FUNCTION_BLOCK MUX_DWORD (* See MUX_ANY *)
  (* Standard: 61131-3 *)
  (* Version 0.0, 2004-12-15, JHC, Rockwell Automation, Converted from SRC format. *)
  (* Compiler header: package fb.rt.plc.select; *)
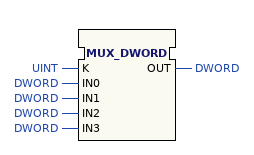
  VAR_INPUT
    K : UINT;
    IN0 : DWORD;
    IN1 : DWORD;
    IN2 : DWORD;
    IN3 : DWORD;
  END_VAR
  VAR_OUTPUT
    OUT : DWORD;
  END_VAR
END_FUNCTION_BLOCK
